PROGRAM MAIN
VAR

END_VAR

END_PROGRAM

(* stored: Version 1.1.0.1, ProductVersion 3.1.4024.0
   POU MAIN: Id {d09ccafb-9881-4e93-b2ee-602c7b940cd3}, SpecialFunc None *)
